// TwinCAT 3 PLC project Automotive
// ProgramVersion: 3.1.4023.0
// libraries:
//   Tc2_MC2, * (Beckhoff Automation GmbH)
//   Tc2_NC, * (Beckhoff Automation GmbH)
//   Tc2_Standard, * (Beckhoff Automation GmbH)
//   Tc2_System, * (Beckhoff Automation GmbH)
//   Tc2_TcpIp, * (Beckhoff Automation GmbH)
//   Tc2_Utilities, * (Beckhoff Automation GmbH)
//   Tc3_Module, * (Beckhoff Automation GmbH)
//   VisuDialogs, * (System)
//   VisuSymbols,3.5.10.0,System
// project tree:
//   Autonoom_POU/ peddal.TcPOU
//   DUTs/ E_State.TcDUT
//   GlobalPOUs/ MAIN.TcPOU, Scaling.TcPOU
//   / GlobalTextList.TcGTLO, PlcTask.TcTTO (not stored), Visualization Manager.TcVMO (not stored)
//   GVLs/ GVL_AxisCtr.TcGVL, GVL_IO.TcGVL, GVL_Lights.TcGVL, GVL_NC.TcGVL (not stored), GVL_SAFETY.TcGVL
//   Motion_POUs/ Command_to_Action.TcPOU, DegreesToRelativeMovment.TcPOU, movements.TcPOU, PositionToDegree.TcPOU (not stored), POUNCPowerOn.TcPOU (not stored), Torque_reading.TcPOU
//   TCPIP_POU/ FB_TcpServer.TcPOU, FnR_Switch.TcPOU, GetSpeedSteer.TcPOU, Lights.TcPOU, RunTCP.TcPOU, SafetyMode.TcPOU, TCPTimeOut.TcPOU
//   VISUs/ ImagePool.TcIPO (not stored), testLights.TcVIS, testStepperVisu.TcVIS
// real-time tasks:
//   TASK PlcTask: cycle T#10ms, priority 21, ADS port 350
// motion (NC):
//   TASK NC-SteeringAxis SAF: cycle T#2ms, priority 4, ADS port 501
//   TASK NC-SteeringAxis SVB: cycle T#10ms, priority 8, ADS port 511
//   AXIS Axis 1 (id 1)
//     OtherSettings: AllowMotionCmdToSlave=true
//     encoder EncType=1
//     drive DrvType=5
//       Analog: TorqueSetpointScale=10, ScaleFactorActTorque=0.1
//       TimeComp: TaskDelayCycles=1
//     controller CtrType=1
//       CtrPara: PriorControlFactor=1
//         Observer: BandWidth=20
// I/O:
//   DEVICE EtherCat (EtherCAT) (disabled), AmsNetId 192.168.0.113.2.1
//     Head Unit(EK1100) [EK1100 EtherCAT Coupler (2A E-Bus)]
//       Safety PLC (EL6900) [EL6900, TwinSAFE PLC]
//       safety input (EL1904) [EL1904, 4 Ch. Safety Input 24V, TwinSAFE]
//         modules: Module 1 (FSOES)
//       Digitale Input (EL1008) [EL1008 8Ch. Dig. Input 24V, 3ms]
//       Digitale Output (EL2008) [EL2008 8Ch. Dig. Output 24V, 0.5A]
//       Analoge Input (EL3062) [EL3062 2Ch. Ana. Input 0-10V]
//       Analoge Output (EL4002) [EL4002 2Ch. Ana. Output 0-10V, 12bit]
// variable links:
//   EtherCat (EtherCAT) <-> EtherCat (EtherCAT)/Head Unit(EK1100)/Safety PLC (EL6900)
//     Head Unit(EK1100)/safety input (EL1904)/Module 1 (FSOES)/RxPDO/FSOE <-> ConnectionInputs/Message_2 TxPDO
//   EtherCat (EtherCAT) <-> EtherCat (EtherCAT)/Head Unit(EK1100)/safety input (EL1904)
//     Head Unit(EK1100)/Safety PLC (EL6900)/ConnectionOutputs/Message_2 RxPDO <-> Module 1 (FSOES)/TxPDO/FSOE
//   Automotive/Automotive Instance <-> EtherCat (EtherCAT)/Head Unit(EK1100)/Safety PLC (EL6900)
//     PlcTask Outputs/GVL_SAFETY.RestartSAFETY <-> StandardOutputs/Standard In Var 1
//   Automotive/Automotive Instance <-> NC-SteeringAxis SAF/Axes/Axis 1
//     PlcTask Inputs/GVL_NC.stXAxis.NcToPlc <-> Outputs/ToPlc
//     PlcTask Outputs/GVL_NC.stXAxis.PlcToNc <-> Inputs/FromPlc

// ---- DUTs/E_State.TcDUT
{attribute 'qualified_only'}
{attribute 'strict'}
TYPE E_State :
(
 	STATE_INIT,
	STATE_CONNECTING,
	STATE_RECEIVING_DATA,
	STATE_SENDING_DATA,
	STATE_PROCESSING_DATA
);
END_TYPE

// ---- GVLs/GVL_AxisCtr.TcGVL
{attribute 'qualified_only'}
VAR_GLOBAL
	bXAxisEnable : BOOL;
	
	
END_VAR

// ---- GVLs/GVL_IO.TcGVL
{attribute 'qualified_only'}
VAR_GLOBAL
	I_bXAxisLimitSwPos AT %I* : BOOL;
	I_bXAxisLimitSwNeg AT %I* : BOOL;
	
	ResetIn AT %I* : BOOL;
END_VAR

// ---- GVLs/GVL_Lights.TcGVL
{attribute 'qualified_only'}
VAR_GLOBAL
//	blinkLeft : BOOL;
//	blinkRight : BOOL;
//	lightFront : BOOL;
//	lightRear : BOOL;
//	lightBrake : BOOL;

	LightsFront 	AT%Q*   : BOOL;
	LightsRear 		AT%Q*  	: BOOL;
	LightsBrake 	AT%Q* 	: BOOL;
	LightsReverse 	AT%Q*  	: BOOL;
    BlinkerLeft 	AT%Q*  	: BOOL;
    BlinkerRight 	AT%Q*  	: BOOL;
END_VAR

// ---- GVLs/GVL_SAFETY.TcGVL
{attribute 'qualified_only'}
VAR_GLOBAL
	RestartSAFETY AT%Q* : BOOL;	
	SafetyTriggerd : BOOL;
	LowMode : BOOL;
END_VAR

// ---- Autonoom_POU/peddal.TcPOU
PROGRAM peddal
VAR
	//autonoom
	Autonoom : BOOL;
	SetAutonoom : BOOL;	
	
	//voor inleen pedal en rem
	RemIngedrukt : BOOL;
	InputNum AT%I* : INT;
	PercentagePedal : REAL;

	//Voor Motion
	fbReadXaxisStatus: MC_ReadStatus;
	triggerAutonoom: F_TRIG;
	LowMode : BOOL;
END_VAR

   triggerAutonoom(CLK:= SetAutonoom, Q=> );
Autonoom S= TriggerAutonoom.Q;
IF Autonoom THEN
	PercentagePedal := Scaling(Input:= InputNum, Imin:= 0, Imax:= 32767, Qmin:= 0, Qmax:= 100);
  Autonoom R= RemIngedrukt OR PercentagePedal > 10;
END_IF

IF LowMode THEN // als lowmode aan is, is maximum throtthe 50%
		IF PercentagePedal > 50 THEN
			PercentagePedal := 50;
		END_IF
END_IF

END_PROGRAM

// ---- GlobalPOUs/Scaling.TcPOU
FUNCTION Scaling : REAL
VAR_INPUT
	Input : INT;
	Imin : REAL;
	Imax : REAL;
	Qmin : REAL;
	Qmax : REAL;
END_VAR
VAR_OUTPUT
END_VAR
VAR
	schaalfactor : REAL;
	offset : REAL;
END_VAR

schaalfactor := (Qmax - Qmin)/(Imax - Imin);
offset := Qmin - (Imin*schaalfactor);
Scaling := (schaalfactor * Input + offset);

END_FUNCTION

// ---- GlobalPOUs/MAIN.TcPOU
PROGRAM MAIN
VAR
	//Voor Motion
	fbReadXaxisStatus: MC_ReadStatus;
	
END_VAR

RunTCP(); //Runs TCP server, lights etc are controlled with this
   peddal();

fbReadXaxisStatus(
	Axis:=GVL_NC.stXAxis , 
	Enable:= GVL_AxisCtr.bXAxisEnable , 
	Valid=> , Busy=> , Error=> , 
	ErrorID=> , ErrorStop=> , 
	Disabled=> , Stopping=> , 
	StandStill=> , DiscreteMotion=> , 
	ContinuousMotion=> , SynchronizedMotion=> , 
	Homing=> , ConstantVelocity=> , 
	Accelerating=> , Decelerating=> , 
	Status=> GVL_NC.stXaxisStatus);
	
	POUNCPowerOn();
	movements();

END_PROGRAM

// ---- TCPIP_POU/RunTCP.TcPOU
PROGRAM RunTCP
VAR
	fbTcpServer 	: FB_TcpServer;
	SrvNetId		: STRING := '';
	ServerAddress 	: STRING := '';
	ServerPort 		: UDINT := 24100;
	
	sResponse		: STRING;
	sCommand		: STRING;
	bBusy			: BOOL;
	err				: BOOL;
	errid			: UDINT;
	
	(*
//	blinkLeft : BOOL;
//	blinkRight : BOOL;
//	lightFront : BOOL;
//	lightRear : BOOL;
//	lightBrake : BOOL;

	LightsFront   : BOOL;
	LightsRear 	: BOOL;
	LightsBrake	: BOOL;
	LightsReverse : BOOL;
    BlinkerLeft     : BOOL;
    BlinkerRight    : BOOL;*)
	
END_VAR

fbTcpServer(
	NetId:= SrvNetId, 
	ServerAdr:= ServerAddress, 
	ServerPort:= ServerPort, 
	sSend := sResponse,
	sReceive=> sCommand, 
	bBusy=> bBusy, 
	err=> err, 
	errid=> errid);
	
	sResponse := sCommand;
	
	TCPTimeOut();
	Lights();
	FnR_Switch();
	SafetyMode();
	GetSpeedSteer();

END_PROGRAM

// ---- TCPIP_POU/FB_TcpServer.TcPOU
FUNCTION_BLOCK FB_TcpServer
VAR_INPUT
	NetId				: STRING; 	(* Server AmsNetId *)
	ServerAdr 			: STRING;	(* Server IP address *)
	ServerPort 			: UDINT;	(* Server port number *)
	sSend 				: STRING;	(* String to be sent *)
END_VAR
VAR_OUTPUT
	sReceive			: STRING;	(* String received *)
	bBusy				: BOOL;
	err					: BOOL;
	errid				: UDINT;
END_VAR
VAR
	fbSocketCloseAll	: FB_SocketCloseAll :=  ( sSrvNetID := '', tTimeout := DEFAULT_ADS_TIMEOUT );
	bCloseAll			: BOOL := TRUE;
		
	Timeout 			: TIME := T#10S;
	fbSocketListen		: FB_SocketListen := (bExecute := TRUE);
	fbSocketReceive		: FB_SocketReceive;
	fbSocketAccept		: FB_SocketAccept;
	fbSocketSend 		: FB_SocketSend;
	hListen				: T_HSOCKET;
	hSocket				: T_HSOCKET;
    
	bConnAccepted		: BOOL;            	
	RxBuffer			: STRING;
	state				: E_State;
           	
	timer				: TON;
	
	
	
	
END_VAR

//https://github.com/vancassa/TwinCAT_TCP_IP_Server/tree/master/Examples/TwinCAT_Program

IF bCloseAll THEN (*On PLC reset or program download close all old connections *)
	bCloseAll := FALSE;
	fbSocketCloseAll( bExecute:= TRUE );
ELSE
	fbSocketCloseAll( bExecute:= FALSE );
END_IF

IF sSend = '' THEN
	sSend := 'Default response';
END_IF
				
timer(IN:= , PT:= T#500MS, Q=> , ET=> );


 
fbSocketListen(
		sSrvNetId:= NetId, 
		sLocalHost:= ServerAdr, 
		nLocalPort:= ServerPort, 
		bExecute:= , 
		tTimeout:= Timeout, 
		bBusy=> bBusy, 
		bError=> err, 
		nErrId=> errid, 
		hListener=> hListen);

fbSocketAccept(
		sSrvNetId:= NetId, 
		hListener:= hListen, 
		bExecute:= , 
		tTimeout:= Timeout, 
		bAccepted=> bConnAccepted, 
		bBusy=> bBusy, 
		bError=> err, 
		nErrId=> errid, 
		hSocket=> hSocket);
	
fbSocketSend(
		sSrvNetId:= NetId, 
		hSocket:= hSocket, 
		cbLen:= LEN(sSend), 
		pSrc:= ADR(sSend), 
		bExecute:= , 
		tTimeout:= Timeout, 
		bBusy=> bBusy, 
		bError=> err, 
		nErrId=> errid);

fbSocketReceive(
		sSrvNetId:= NetId, 
		hSocket:= hSocket, 
		cbLen:= SIZEOF(RxBuffer), 
		pDest:= ADR(RxBuffer), 
		bExecute:= , 
		tTimeout:= Timeout, 
		bBusy=> bBusy, 
		bError=> err, 
		nErrId=> errid, 
		nRecBytes=> );
		
CASE state OF
	E_State.STATE_INIT:
		//Open the port
		fbSocketListen.bExecute := TRUE;
		state := E_State.STATE_CONNECTING;
		
		
	E_State.STATE_CONNECTING:
		fbSocketListen.bExecute := FALSE;
		//Accept incoming connection every half a second
		IF NOT fbSocketListen.bBusy AND NOT fbSocketListen.bError THEN
			fbSocketAccept.bExecute := FALSE;
			timer.IN := TRUE;
	
			IF bConnAccepted THEN
				fbSocketReceive.bExecute := TRUE;
				state := E_State.STATE_RECEIVING_DATA;
			ELSIF timer.Q THEN
				fbSocketAccept.bExecute := TRUE;
				timer.IN := FALSE;
			END_IF
		END_IF
	
		
	E_State.STATE_RECEIVING_DATA:
		fbSocketReceive.bExecute := FALSE;
		
		IF NOT fbSocketReceive.bBusy AND NOT fbSocketReceive.bError THEN
			IF fbSocketReceive.nRecBytes = 0 THEN
				//if there's no data received, reset the fbSocketReceive
				fbSocketReceive.bExecute := TRUE;
			ELSE
				MEMSET(ADR(sReceive),0,SIZEOF(sReceive));
				MEMCPY(ADR(sReceive), fbSocketReceive.pDest, fbSocketReceive.nRecBytes);
				

				fbSocketSend.bExecute := TRUE;
				state := E_State.STATE_SENDING_DATA;
			END_IF
		END_IF
	
		
	E_State.STATE_SENDING_DATA:
		fbSocketSend.bExecute := FALSE;
		
		IF NOT fbSocketSend.bBusy AND NOT fbSocketSend.bError THEN 
				fbSocketReceive.bExecute := TRUE;
				state := E_State.STATE_RECEIVING_DATA;
		END_IF
END_CASE

END_FUNCTION_BLOCK

// ---- TCPIP_POU/TCPTimeOut.TcPOU
PROGRAM TCPTimeOut
VAR
	fbLocalTime : FB_LocalSystemTime;
	iPreviousTime : WORD := 0;
END_VAR


fbLocalTime(
	sNetId := ,
	bEnable := TRUE,
	dwCycle := 10,
	dwOpt := ,
	tTimeout := DEFAULT_ADS_TIMEOUT,
);

	IF fbLocalTime.systemTime.wMilliseconds - iPreviousTime >= 200 THEN	
		GVL_SAFETY.SafetyTriggerd := TRUE;	
	END_IF
	
	IF RunTCP.sCommand > '' THEN
		iPreviousTime := fbLocalTime.systemTime.wMilliseconds;
	END_IF

END_PROGRAM

// ---- TCPIP_POU/Lights.TcPOU
PROGRAM Lights
VAR
END_VAR

IF RunTCP.sCommand = 'BL1' THEN	//blinker left on	//These are connected to the blinker relay, so only high signal suffices
    GVL_Lights.BlinkerLeft    := TRUE;
    GVL_Lights.BlinkerRight   := FALSE;
ELSIF RunTCP.sCommand = 'BL0' THEN	//blinker left off
    GVL_Lights.BlinkerLeft    := FALSE;
    GVL_Lights.BlinkerRight := FALSE;
ELSIF RunTCP.sCommand = 'BR1' THEN	//blinker right on
    GVL_Lights.BlinkerRight   := TRUE;
    GVL_Lights.BlinkerLeft    := FALSE;
ELSIF RunTCP.sCommand = 'BR0' THEN	//blinker right off
    GVL_Lights.BlinkerRight  := FALSE;
    GVL_Lights.BlinkerLeft   := FALSE;
ELSIF RunTCP.sCommand = 'L1' THEN //lights on
	GVL_Lights.LightsFront := TRUE;
	GVL_Lights.LightsRear := TRUE;
ELSIF RunTCP.sCommand = 'L0' THEN	//lights off
	GVL_Lights.LightsFront := FALSE;
	GVL_Lights.LightsRear := FALSE;
	//TODO link to reverse
(*ELSIF RunTCP.sCommand = 'ron' THEN	//reverse light on
	GVL_Lights.LightsReverse := TRUE;
ELSIF RunTCP.sCommand = 'roff' THEN	//reverse light off
	GVL_Lights.LightsReverse := FALSE;*)
ELSIF RunTCP.sCommand = 'B1' THEN	//brake light on
	GVL_Lights.LightsBrake := TRUE;
ELSIF RunTCP.sCommand = 'B0' THEN	//brake light off
	GVL_Lights.LightsBrake := FALSE;
ELSE
    GVL_Lights.BlinkerRight := FALSE;
    GVL_Lights.BlinkerLeft  := FALSE;

END_IF

END_PROGRAM

// ---- TCPIP_POU/FnR_Switch.TcPOU
PROGRAM FnR_Switch
VAR
	qFNR : BOOL; //0 = user control, 1 = PLC controlled FNR
	qFNRDir : BOOL; //Sets direction 0 = reverse, 1 = forward
END_VAR

//Program to select what direction the car should go
IF RunTCP.sCommand = 'F' THEN //Forward mode
	qFNR := TRUE;
	qFNRDir := TRUE;
ELSIF RunTCP.sCommand = 'R' THEN //Reverse mode
	qFNR := TRUE;
	qFNRDir := FALSE;
ELSIF RunTCP.sCommand = 'M' THEN //supposed to be manual mode
	qFNR := FALSE;
	qFNRDir := FALSE; //This one doesn't really matter
END_IF

END_PROGRAM

// ---- TCPIP_POU/SafetyMode.TcPOU
PROGRAM SafetyMode
VAR
	
END_VAR

IF RunTCP.sCommand = 'HIGHMODE' THEN
	GVL_SAFETY.LowMode := FALSE;
ELSIF RunTCP.sCommand = 'LOWMODE' THEN
	GVL_SAFETY.LowMode := TRUE;
END_IF

END_PROGRAM

// ---- TCPIP_POU/GetSpeedSteer.TcPOU
PROGRAM GetSpeedSteer
VAR
	steerString : STRING;
	pedalString : STRING;
	bExecuteSteer : BOOL;
END_VAR

//bExecuteSteer := FALSE;

IF movements.Command_to_Action_0.Busy THEN
	bExecuteSteer := FALSE;
END_IF

IF FIND(STR1:= 'Steer', STR2:= RunTCP.sCommand) = 1 THEN
	steerString := RunTCP.sCommand;
	bExecuteSteer := TRUE;
ELSIF FIND(STR1:= 'Throttle', STR2:= RunTCP.sCommand) = 1 THEN
	pedalString := RunTCP.sCommand;
END_IF

END_PROGRAM

// ---- Motion_POUs/movements.TcPOU
PROGRAM movements
VAR
	MC_MoveAbsolute_0: MC_MoveAbsolute;
	ExecuteMovement : BOOL;
	
	movementBuffer : MC_BufferMode; 
	
	DegreesToRelativeMovment_0: DegreesToRelativeMovment;
	
	Command_to_Action_0: Command_to_Action;
	
	PositionToDegree_0: PositionToDegree;
END_VAR

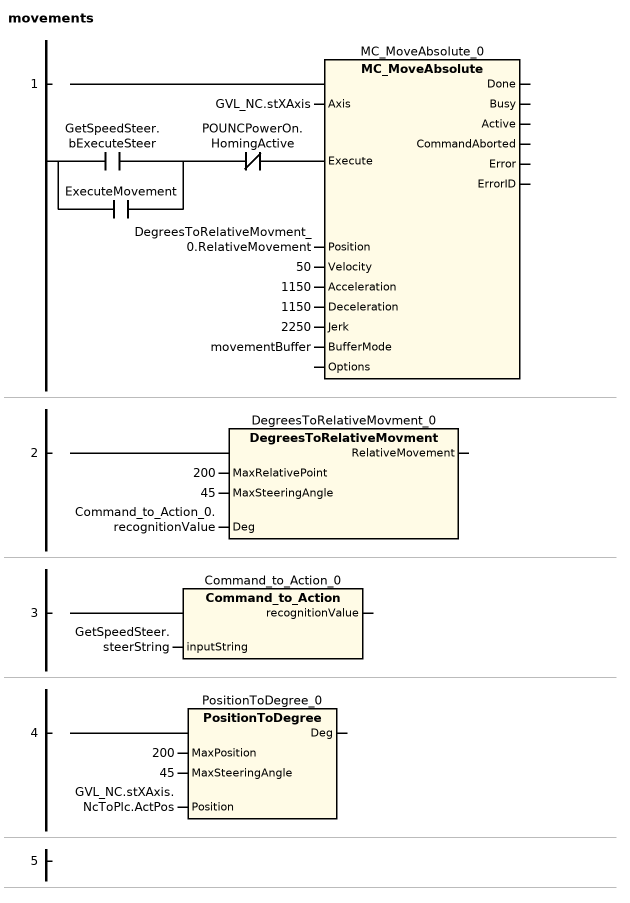
// NETWORK 1
MC_MoveAbsolute_0(
    Axis := GVL_NC.stXAxis,
    Execute := (GetSpeedSteer.bExecuteSteer OR ExecuteMovement) AND NOT POUNCPowerOn.HomingActive,
    Position := DegreesToRelativeMovment_0.RelativeMovement,
    Velocity := 50,
    Acceleration := 1150,
    Deceleration := 1150,
    Jerk := 2250,
    BufferMode := movementBuffer); // MC_MoveAbsolute

// NETWORK 2
DegreesToRelativeMovment_0(
    MaxRelativePoint := 200,
    MaxSteeringAngle := 45,
    Deg := Command_to_Action_0.recognitionValue); // DegreesToRelativeMovment

// NETWORK 3
Command_to_Action_0(inputString := GetSpeedSteer.steerString); // Command_to_Action

// NETWORK 4
PositionToDegree_0(MaxPosition := 200, MaxSteeringAngle := 45, Position := GVL_NC.stXAxis.NcToPlc.ActPos); // PositionToDegree

// NETWORK 5

END_PROGRAM

// ---- Motion_POUs/DegreesToRelativeMovment.TcPOU
FUNCTION_BLOCK DegreesToRelativeMovment
VAR_INPUT
	MaxRelativePoint : LREAL;
	MaxSteeringAngle : INT;
	Deg : LREAL;
END_VAR
VAR_OUTPUT
	RelativeMovement : LREAL;
END_VAR
VAR
END_VAR

IF (Deg > 0 OR Deg < 0) THEN
	RelativeMovement := (MaxRelativePoint/MaxSteeringAngle)*Deg;
ELSIF (Deg = 0) THEN
	RelativeMovement := 0;		
END_IF

END_FUNCTION_BLOCK

// ---- Motion_POUs/Command_to_Action.TcPOU
FUNCTION_BLOCK Command_to_Action
VAR_INPUT
	inputString : STRING;
END_VAR
VAR_OUTPUT
	recognitionValue : REAL;
	Busy : BOOL;
END_VAR
VAR
	putString : STRING;
	recognitionString : STRING := 'Steer(';
	stringLength : int;
END_VAR

inputString := GetSpeedSteer.steerString;

Busy := FALSE;
IF GetSpeedSteer.bExecuteSteer THEN
	Busy := TRUE;
END_IF

IF FIND(STR1:= inputString  , STR2:= recognitionString ) = 1 THEN
	putString := DELETE(STR:=inputString , LEN:= 6 , POS:=1 );
	stringLength := LEN(putstring);
	putString := DELETE(STR:=putString , LEN:= 1 , POS:= stringLength);
	recognitionValue := STRING_TO_INT(putString);
END_IF

END_FUNCTION_BLOCK

// ---- Motion_POUs/Torque_reading.TcPOU
PROGRAM Torque_reading
VAR
	MC_TorqueControl_0: MC_TorqueControl;
END_VAR

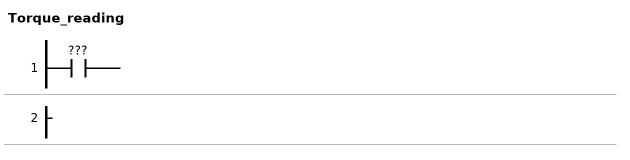
// NETWORK 1

// NETWORK 2

END_PROGRAM

// ---- GlobalTextList.TcGTLO
TEXTLIST GlobalTextList
  163 = '%10.1f'
  781 = '%1f'
  35 = '%d'
  559 = '%d s'
  953 = '%i'
  523 = 'EndSwitch'
  895 = 'Execute'
  52 = 'Reset'
  627 = 'setAngle'
  485 = 'Start Homing'
  860 = 'StartHoming'
  447 = 'X-Axis enable'
  34 = 'x-axis limit+'
  942 = 'x-axis limit-'
END_TEXTLIST

// ---- VISUs/testLights.TcVIS
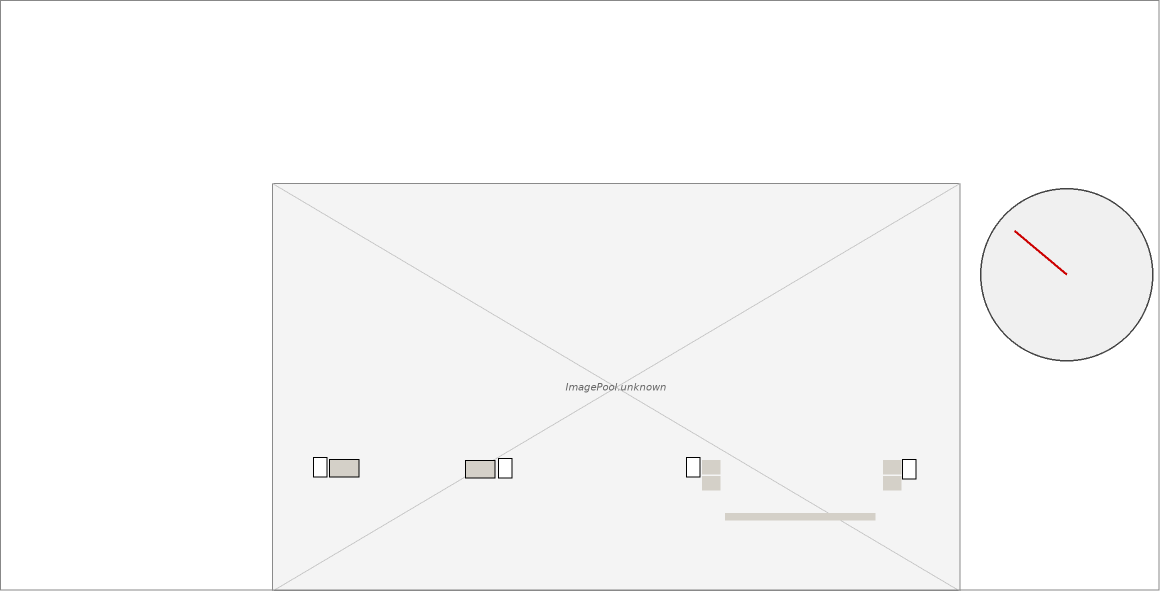
VISUALIZATION testLights  // 1160x591
    Image (272,183 688x408), image: ImagePool.unknown
    RoundedRectangle (498,458 14x20), colour toggle: GVL_Lights.BlinkerLeft
    RoundedRectangle (313,457 14x20), colour toggle: GVL_Lights.BlinkerRight
    RoundedRectangle (465,460 30x18), colour toggle: GVL_Lights.LightsFront
    RoundedRectangle (686,457 14x20), colour toggle: GVL_Lights.BlinkerLeft
    RoundedRectangle (902,459 14x20), colour toggle: GVL_Lights.BlinkerRight
    RoundedRectangle (329,459 30x18), colour toggle: GVL_Lights.LightsFront
    RoundedRectangle (702,460 18x14), colour toggle: GVL_Lights.LightsRear
    RoundedRectangle (702,476 18x14), colour toggle: GVL_Lights.LightsBrake
    RoundedRectangle (883,460 18x14), colour toggle: GVL_Lights.LightsRear
    RoundedRectangle (883,476 18x14), colour toggle: GVL_Lights.LightsBrake
    RoundedRectangle (725,513 150x7), colour toggle: GVL_Lights.LightsReverse
    Meter90 (973,188 187x173), value: movements.PositionToDegree_0.Deg, style: Meter-Meter90-Gray, scale format: %.1f, scale -45..45
END_VISUALIZATION

// ---- VISUs/testStepperVisu.TcVIS
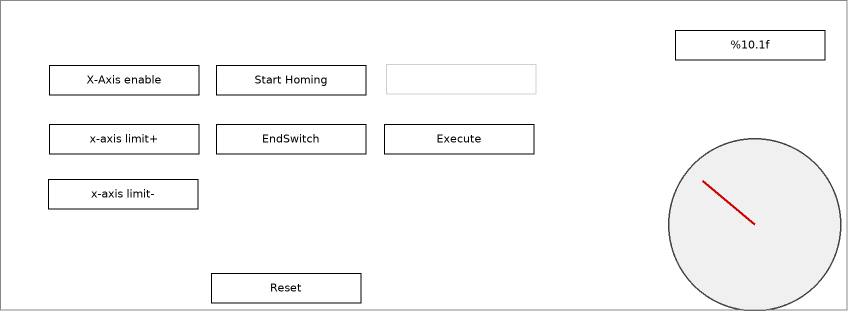
VISUALIZATION testStepperVisu  // 848x311
    Rectangle (49,65 150x30), "X-Axis enable"
        toggle GVL_AxisCtr.bXAxisEnable
    RoundedRectangle (49,124 150x30), "x-axis limit+", colour toggle: GVL_IO.I_bXAxisLimitSwPos
        toggle GVL_IO.I_bXAxisLimitSwPos
    RoundedRectangle (48,179 150x30), "x-axis limit-", colour toggle: GVL_IO.I_bXAxisLimitSwNeg
        toggle GVL_IO.I_bXAxisLimitSwNeg
    Rectangle (675,30 150x30), "%10.1f", text variable: GVL_NC.stXAxis.NcToPlc.ActPos
    Rectangle (384,124 150x30), "Execute"
        tap movements.ExecuteMovement
    Rectangle (216,65 150x30), "Start Homing"
        tap POUNCPowerOn.StartHoming
    Rectangle (216,124 150x30), "EndSwitch"
        toggle POUNCPowerOn.endSW
    Rectangle (211,273 150x30), "Reset"
        tap POUNCPowerOn.reset
    Meter90 (661,138 187x173), value: movements.PositionToDegree_0.Deg, style: Meter-Meter90-Gray, scale format: %.1f, scale -45..45
    Textfield (386,64 150x30), text variable: movements.Command_to_Action_0.inputString
        OnMouseDown: write the text variable via Default
END_VISUALIZATION
